FUNCTION TFValutaFormatureMultipleAttivate : BOOL // Valuta se ci sono più formature DIVERSE attive 
VAR_INPUT
	Forming : POINTER TO ARRAY [1..MAXFORMING] OF TFMachinePalletizer_Forming; //Struttura formature
END_VAR
VAR
	f : INT;	// Indice formatura
	c: INT;
	TFValutaFormatureMultipleAttivateMEM: BOOL;
END_VAR
// Valuta se ci sono più formature DIVERSE attive

// Valuta se ci sono più formature DIVERSE attive 
FOR f := 1 TO 4 DO
	CASE f OF
		1:
			IF Forming^[f].Enable = 1 THEN					// se la formatura è abilitata
				IF Forming^[2].Enable = 1 THEN
					IF Forming^[f].GUID <> Forming^[2].GUID THEN //Se la formatura attiva è diversa da quella su indice i
						FOR c := 1 TO MAXFORMINGCODE DO
							IF Forming^[f].Code[c] > 0 THEN //Se ha almeno un codice assegnato
								TFValutaFormatureMultipleAttivateMEM := TRUE;
								//RETURN;
							END_IF
							IF Forming^[2].Code[c] > 0 AND TFValutaFormatureMultipleAttivateMEM THEN //Se ha almeno un codice assegnato
								TFValutaFormatureMultipleAttivate := TRUE;
								RETURN;
							ELSE
								TFValutaFormatureMultipleAttivate := FALSE;
								//RETURN;
							END_IF
						END_FOR
					END_IF
				END_IF	
				IF Forming^[3].Enable = 1 THEN
					IF Forming^[f].GUID <> Forming^[3].GUID THEN //Se la formatura attiva è diversa da quella su indice i
						FOR c := 1 TO MAXFORMINGCODE DO
							IF Forming^[f].Code[c] > 0 THEN //Se ha almeno un codice assegnato
								TFValutaFormatureMultipleAttivateMEM := TRUE;
								//RETURN;
							END_IF
							IF Forming^[3].Code[c] > 0 AND TFValutaFormatureMultipleAttivateMEM THEN //Se ha almeno un codice assegnato
								TFValutaFormatureMultipleAttivate := TRUE;
								RETURN;
							ELSE
								TFValutaFormatureMultipleAttivate := FALSE;
								//RETURN;
							END_IF
						END_FOR
					END_IF
				END_IF
				IF Forming^[4].Enable = 1 THEN
					IF Forming^[f].GUID <> Forming^[4].GUID THEN
						FOR c := 1 TO MAXFORMINGCODE DO
							IF Forming^[f].Code[c] > 0 THEN
								TFValutaFormatureMultipleAttivateMEM := TRUE;
								//RETURN;
							END_IF
							IF Forming^[4].Code[c] > 0 AND TFValutaFormatureMultipleAttivateMEM THEN //Se ha almeno un codice assegnato
								TFValutaFormatureMultipleAttivate := TRUE;
								RETURN;
							ELSE
								TFValutaFormatureMultipleAttivate := FALSE;
								//RETURN;
							END_IF
						END_FOR
					END_IF
				END_IF 
			END_IF
		2:
			IF Forming^[f].Enable = 1 THEN					// se la formatura è abilitata
				IF Forming^[1].Enable = 1 THEN
					IF Forming^[f].GUID <> Forming^[1].GUID THEN
						FOR c := 1 TO MAXFORMINGCODE DO
							IF Forming^[f].Code[c] > 0 THEN
								TFValutaFormatureMultipleAttivateMEM := TRUE;
								//RETURN;
							END_IF
							IF Forming^[1].Code[c] > 0 AND TFValutaFormatureMultipleAttivateMEM THEN //Se ha almeno un codice assegnato
								TFValutaFormatureMultipleAttivate := TRUE;
								RETURN;
							ELSE
								TFValutaFormatureMultipleAttivate := FALSE;
								//RETURN;
							END_IF
						END_FOR
					END_IF
				END_IF
				IF Forming^[3].Enable = 1 THEN
					IF Forming^[f].GUID <> Forming^[3].GUID THEN //Se la formatura attiva è diversa da quella su indice i
						FOR c := 1 TO MAXFORMINGCODE DO
							IF Forming^[f].Code[c] > 0 THEN //Se ha almeno un codice assegnato
								TFValutaFormatureMultipleAttivateMEM := TRUE;
								//RETURN;
							END_IF
							IF Forming^[3].Code[c] > 0 AND TFValutaFormatureMultipleAttivateMEM THEN //Se ha almeno un codice assegnato
								TFValutaFormatureMultipleAttivate := TRUE;
								RETURN;
							ELSE
								TFValutaFormatureMultipleAttivate := FALSE;
								//RETURN;
							END_IF
						END_FOR
					END_IF
				END_IF
				IF Forming^[4].Enable = 1 THEN
					IF Forming^[f].GUID <> Forming^[4].GUID THEN
						FOR c := 1 TO MAXFORMINGCODE DO
							IF Forming^[f].Code[c] > 0 THEN
								TFValutaFormatureMultipleAttivateMEM := TRUE;
								//RETURN;
							END_IF
							IF Forming^[4].Code[c] > 0 AND TFValutaFormatureMultipleAttivateMEM THEN //Se ha almeno un codice assegnato
								TFValutaFormatureMultipleAttivate := TRUE;
								RETURN;
							ELSE
								TFValutaFormatureMultipleAttivate := FALSE;
								//RETURN;
							END_IF
						END_FOR
					END_IF
				END_IF 
			END_IF
		3:
			IF Forming^[f].Enable = 1 THEN					// se la formatura è abilitata
				IF Forming^[1].Enable = 1 THEN
					IF Forming^[f].GUID <> Forming^[1].GUID THEN
						FOR c := 1 TO MAXFORMINGCODE DO
							IF Forming^[f].Code[c] > 0 THEN
								TFValutaFormatureMultipleAttivateMEM := TRUE;
								//RETURN;
							END_IF
							IF Forming^[1].Code[c] > 0 AND TFValutaFormatureMultipleAttivateMEM THEN //Se ha almeno un codice assegnato
								TFValutaFormatureMultipleAttivate := TRUE;
								RETURN;
							ELSE
								TFValutaFormatureMultipleAttivate := FALSE;
								//RETURN;
							END_IF
						END_FOR
					END_IF
				END_IF
				IF Forming^[2].Enable = 1 THEN
					IF Forming^[f].GUID <> Forming^[2].GUID THEN //Se la formatura attiva è diversa da quella su indice i
						FOR c := 1 TO MAXFORMINGCODE DO
							IF Forming^[f].Code[c] > 0 THEN //Se ha almeno un codice assegnato
								TFValutaFormatureMultipleAttivateMEM := TRUE;
								//RETURN;
							END_IF
							IF Forming^[2].Code[c] > 0 AND TFValutaFormatureMultipleAttivateMEM THEN //Se ha almeno un codice assegnato
								TFValutaFormatureMultipleAttivate := TRUE;
								RETURN;
							ELSE
								TFValutaFormatureMultipleAttivate := FALSE;
								//RETURN;
							END_IF
						END_FOR
					END_IF
				END_IF
				IF Forming^[4].Enable = 1 THEN
					IF Forming^[f].GUID <> Forming^[4].GUID THEN
						FOR c := 1 TO MAXFORMINGCODE DO
							IF Forming^[f].Code[c] > 0 THEN
								TFValutaFormatureMultipleAttivateMEM := TRUE;
								//RETURN;
							END_IF
							IF Forming^[4].Code[c] > 0 AND TFValutaFormatureMultipleAttivateMEM THEN //Se ha almeno un codice assegnato
								TFValutaFormatureMultipleAttivate := TRUE;
								RETURN;
							ELSE
								TFValutaFormatureMultipleAttivate := FALSE;
								//RETURN;
							END_IF
						END_FOR
					END_IF
				END_IF 
			END_IF
		4:
			IF Forming^[f].Enable = 1 THEN					// se la formatura è abilitata
				IF Forming^[1].Enable = 1 THEN
					IF Forming^[f].GUID <> Forming^[1].GUID THEN
						FOR c := 1 TO MAXFORMINGCODE DO
							IF Forming^[f].Code[c] > 0 THEN
								TFValutaFormatureMultipleAttivateMEM := TRUE;
								//RETURN;
							END_IF
							IF Forming^[1].Code[c] > 0 AND TFValutaFormatureMultipleAttivateMEM THEN //Se ha almeno un codice assegnato
								TFValutaFormatureMultipleAttivate := TRUE;
								RETURN;
							ELSE
								TFValutaFormatureMultipleAttivate := FALSE;
								//RETURN;
							END_IF
						END_FOR
					END_IF
				END_IF
				IF Forming^[2].Enable = 1 THEN
					IF Forming^[f].GUID <> Forming^[2].GUID THEN
						FOR c := 1 TO MAXFORMINGCODE DO
							IF Forming^[f].Code[c] > 0 THEN
								TFValutaFormatureMultipleAttivateMEM := TRUE;
								//RETURN;
							END_IF
							IF Forming^[2].Code[c] > 0 AND TFValutaFormatureMultipleAttivateMEM THEN //Se ha almeno un codice assegnato
								TFValutaFormatureMultipleAttivate := TRUE;
								RETURN;
							ELSE
								TFValutaFormatureMultipleAttivate := FALSE;
								//RETURN;
							END_IF
						END_FOR
					END_IF
				END_IF
				IF Forming^[3].Enable = 1 THEN
					IF Forming^[f].GUID <> Forming^[3].GUID THEN
						FOR c := 1 TO MAXFORMINGCODE DO
							IF Forming^[f].Code[c] > 0 THEN
								TFValutaFormatureMultipleAttivateMEM := TRUE;
								//RETURN;
							END_IF
							IF Forming^[3].Code[c] > 0 AND TFValutaFormatureMultipleAttivateMEM THEN //Se ha almeno un codice assegnato
								TFValutaFormatureMultipleAttivate := TRUE;
								RETURN;
							ELSE
								TFValutaFormatureMultipleAttivate := FALSE;
								//RETURN;
							END_IF
						END_FOR
					END_IF
				END_IF 
			END_IF
		
	END_CASE
END_FOR
TFValutaFormatureMultipleAttivate := FALSE;

END_FUNCTION

(* stored: Version 1.1.0.1, ProductVersion 3.1.4024.11
   POU TFValutaFormatureMultipleAttivate: Id {5021cc4c-b76d-4dc2-9cd2-01aeb97d5779}, SpecialFunc None *)
